TYPE ST_HIERARCHYDATAPK :
STRUCT
	UNITQTY		:STRING;
	GTIN		:STRING;
	EAN			:STRING;
END_STRUCT
END_TYPE

(* stored: Version 1.1.0.1, ProductVersion 3.1.4024.13
   DUT ST_HIERARCHYDATAPK: Id {3189ebcd-f506-4717-bdb8-c8f8cda5cf73} *)
